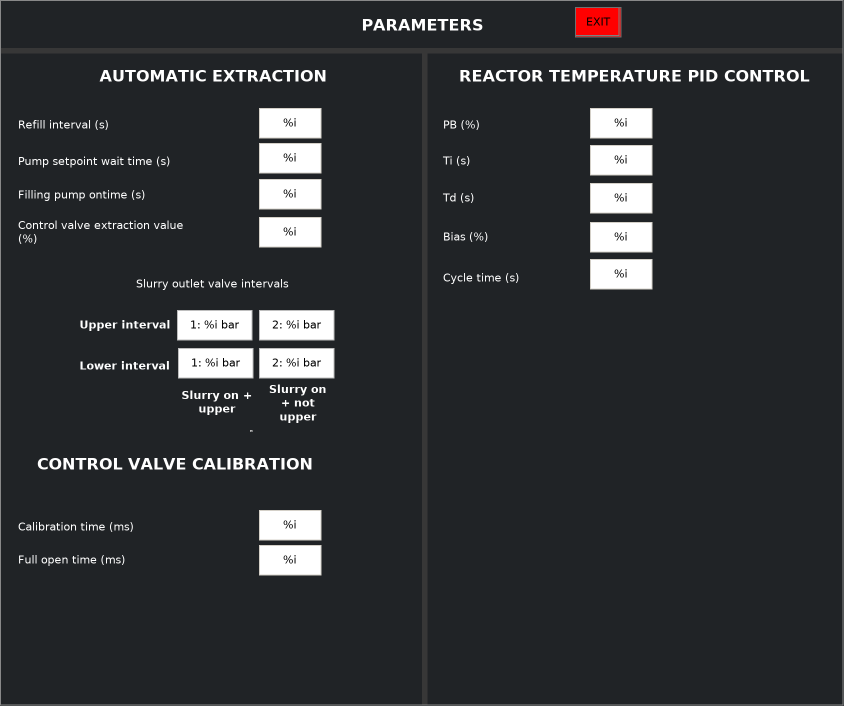
VISUALIZATION ParameterView  // 844x706
    Textfield (259,108 62x30), "%i", text variable: ParameterViewBindings.refillIntervalTextField_TextVariable
        OnMouseDown: write the text variable via VisuDialogs.Numpad, min 1, max 999
    Label (15,103 190x44), "Refill interval (s)"
    Button (575,7 46x30), "EXIT", pressed state: NOT MainScreenBindings.autoExtractionParameterMenuButton_ToggleVariable
        toggle MainScreenBindings.autoExtractionParameterMenuButton_ToggleVariable
    Label (15,173 190x44), "Filling pump ontime (s)"
    Label (15,210 190x44), "Control valve extraction value (%)"
    Textfield (259,179 62x30), "%i", text variable: ParameterViewBindings.pumpOnTimeTextField_TextVariable
        OnMouseDown: write the text variable via VisuDialogs.Numpad, min 1, max 5999
    Textfield (259,217 62x30), "%i", text variable: ParameterViewBindings.controlValveOpeningValueTextField_TextVariable
        OnMouseDown: write the text variable via VisuDialogs.Numpad, min 1, max 5999
    Label (15,139 190x45), "Pump setpoint wait time (s)"
    Textfield (259,143 62x30), "%i", text variable: ParameterViewBindings.pumpSetpointWaitTimeTextField_TextVariable
        OnMouseDown: write the text variable via VisuDialogs.Numpad, min 0, max 999
    Image (250,430 2x1), image: VisuSymbols.Symbols.ArrowBoldRight
    Label (75,303 100x44), "Upper interval"
    Label (75,344 100x44), "Lower interval"
    Textfield (177,310 75x30), "1: %i bar", text variable: MainScreenBindings.UpperIntervalSlurryOnUpperTextField_TextVariable
        OnMouseDown: write the text variable via VisuDialogs.Numpad, min -100, max 100
    Textfield (259,310 75x30), "2: %i bar", text variable: MainScreenBindings.UpperIntervalSlurryOnNotUpperTextField_TextVariable
        OnMouseDown: write the text variable via VisuDialogs.Numpad, min -100, max 100
    Textfield (178,348 75x30), "1: %i bar", text variable: MainScreenBindings.LowerIntervalSlurryOnUpperTextField_TextVariable
        OnMouseDown: write the text variable via VisuDialogs.Numpad, min -100, max 100
    Textfield (259,348 75x30), "2: %i bar", text variable: MainScreenBindings.LowerIntervalSlurryOnNotUpperTextField_TextVariable
        OnMouseDown: write the text variable via VisuDialogs.Numpad, min -100, max 100
    Label (178,380 78x44), "Slurry on + upper"
    Label (262,381 72x44), "Slurry on + not upper"
    Label (5,262 415x44), "Slurry outlet valve intervals"
    Textfield (590,108 62x30), "%i", text variable: ParameterViewBindings.PbTextField_TextVariable
        OnMouseDown: write the text variable via VisuDialogs.Numpad, min 1, max 999
    Label (440,103 103x44), "PB (%)"
    Label (440,139 103x44), "Ti (s)"
    Label (440,176 103x44), "Td (s)"
    Textfield (590,145 62x30), "%i", text variable: ParameterViewBindings.TiTextField_TextVariable
        OnMouseDown: write the text variable via VisuDialogs.Numpad, min 1, max 5999
    Textfield (590,183 62x30), "%i", text variable: ParameterViewBindings.TdTextField_TextVariable
        OnMouseDown: write the text variable via VisuDialogs.Numpad, min 1, max 5999
    Label (440,215 103x44), "Bias (%)"
    Textfield (590,222 62x30), "%i", text variable: ParameterViewBindings.BiasTextField_TextVariable
        OnMouseDown: write the text variable via VisuDialogs.Numpad, min 0, max 999
    Textfield (590,259 62x30), "%i", text variable: ParameterViewBindings.IterationTimeTextField_TextVariable
        OnMouseDown: write the text variable via VisuDialogs.Numpad, min 1, max 5999
    Textfield (259,510 62x30), "%i", text variable: ParameterViewBindings.calibrationTimeTextField_TextVariable
        OnMouseDown: write the text variable via VisuDialogs.Numpad, min 1, max 999999
    Label (15,505 190x44), "Calibration time (ms)"
    Textfield (259,545 62x30), "%i", text variable: ParameterViewBindings.fullOpenTimeTextField_TextVariable
        OnMouseDown: write the text variable via VisuDialogs.Numpad, min 0, max 999999
    Label (15,538 190x44), "Full open time (ms)"
    Label (4,61 419x30), "AUTOMATIC EXTRACTION"
    Label (34,449 321x30), "CONTROL VALVE CALIBRATION"
    Rectangle (422,50 5x655)
    Label (430,61 409x30), "REACTOR TEMPERATURE PID CONTROL"
    Label (264,10 317x30), "PARAMETERS"
    Label (440,256 117x44), "Cycle time (s)"
    Rectangle (1,48 842x5)
END_VISUALIZATION

(* stored: Version 1.1.0.1, ProductVersion 3.1.4024.9
   Visu ParameterView: Id {800908a7-96e7-46b1-b2c8-3866ec22bff5} *)
